// TIA Portal V20 export
DATA_BLOCK "Config"   // DB100
// stored: MemoryReserve 100, Namespace Unit1.Em10
   VAR
      em : "LAF_typeEmConfiguration";   // Configuration of EM Parameters
      cmLaserMarkJRDetect : "LBC_typeDigitalSignalConfiguration";
      cmLaserMarkStageLiftUpDown : "LBC_typeTwoWayActuatorConfiguration";
      cmLaserMarkCoverUpDown : "LBC_typeTwoWayActuatorConfiguration";
      cmLaserMarkControl : "LER_typeLaserMarkConfiguration";
      cmQrFixReaderControl : "LER_typeSRX300Configuration";
   END_VAR
BEGIN
   em.referenceDesignator.parent := WSTRING#'U1';
   em.referenceDesignator.relative := WSTRING#'EM0';
   cmLaserMarkStageLiftUpDown.referenceDesignator := WSTRING#'MARKING STAGE LIFT';
   cmLaserMarkCoverUpDown.referenceDesignator := WSTRING#'LASER MARKING COVER';
   cmLaserMarkControl.hwID.machineStatusID := 363;
   cmLaserMarkControl.hwID.functionStatusID := 364;
   cmLaserMarkControl.hwID.completionStatusID := 365;
   cmLaserMarkControl.hwID.errorStatusID := 366;
   cmLaserMarkControl.hwID.errorCodesID := 367;
   cmLaserMarkControl.hwID.operateParameterID := 368;
   cmLaserMarkControl.hwID."2DCReadResultID" := 369;
   cmLaserMarkControl.hwID.countResultDataID := 370;
   cmLaserMarkControl.hwID.resultDataID := 371;
   cmLaserMarkControl.hwID.generalRequestID := 372;
   cmLaserMarkControl.hwID.functionRequestID := 373;
   cmLaserMarkControl.hwID.requestCompletionClearID := 374;
   cmLaserMarkControl.hwID.requestParameterID := 375;
   cmLaserMarkControl.hwID.requestDataID := 376;
   cmQrFixReaderControl.hwID.handshakeGeneralErrorStatusHwId := 1007;
   cmQrFixReaderControl.hwID.busyStatusHwId := 1006;
   cmQrFixReaderControl.hwID.completionStatusHwId := 1005;
   cmQrFixReaderControl.hwID.errorStatusHwId := 1004;
   cmQrFixReaderControl.hwID.terminalStatusHwId := 1003;
   cmQrFixReaderControl.hwID.unstableReadStatusHwId := 1002;
   cmQrFixReaderControl.hwID.matchingAndGradeStatusHwId := 1001;
   cmQrFixReaderControl.hwID.operationResultStatusHwId := 1000;
   cmQrFixReaderControl.hwID.readDataHeaderHwId := 999;
   cmQrFixReaderControl.hwID.readDataExtendedPart1HwId := 999;
   cmQrFixReaderControl.hwID.readDataExtendedPart2HwId := 999;
   cmQrFixReaderControl.hwID.readDataExtendedPart3HwId := 999;
   cmQrFixReaderControl.hwID.latchErrorClearControlHwId := 998;
   cmQrFixReaderControl.hwID.operationInstructionControlHwId := 997;
   cmQrFixReaderControl.hwID.completionClearControlHwId := 996;
   cmQrFixReaderControl.hwID.parameterBankNumberHwId := 995;
   cmQrFixReaderControl.hwID.userDataHwId := 994;
   cmQrFixReaderControl.triggertime := T#100ms;
   cmQrFixReaderControl.cycleTime := T#1000ms;
END_DATA_BLOCK
